(* CODESYS project cr710siowrapper_RECOVERED_2026-03-05T12-49-56.project
   Company: ifm electronic
   Description: Project template with CR711S configured 2.25MByte Standard 2.25MByte Safety
   Title: ifmCR711S_TemplateProject
   Version: 2.4.10.0

Project tree, tasks and I/O mapping:
  StandardPLC : CR710S Standard, ifm electronic, order no. CR710S, version 3.2.0.0
    application Application
      libraries: ifmR360-3, 1.1.1.0 (ifm electronic); Util, * (System); Standard, * (System); CR710S IOWrapper, 1.0.4.9 (ifm electronic)
      task Task (cyclic, interval t#10ms, priority 0) calls PLC_PRG, HeartBeat
      visualisation SimpleStateSwitch
      EVC
      program CR710S_Config [ST]: config_outputs, config_outgroups, config_inputs
      data type EStates
      program PLC_PRG [ST]
      data type EStation
      global variables GVL_HeartBeat
      program HeartBeat [LD]
    HMI : HMI, ifm electronic, version 3.2.0.0
      User_LEDs : User_LEDs, ifm electronic, version 3.2.0.0
          input  UserLED0_I : LED_IEC_B_INPUT_MAPPING_TYPE  // UserLED0_I
          input  UserLED1_I : LED_IEC_B_INPUT_MAPPING_TYPE  // UserLED1_I
          input  UserLED2_I : LED_IEC_B_INPUT_MAPPING_TYPE  // UserLED2_I
          input  UserLED3_I : LED_IEC_B_INPUT_MAPPING_TYPE  // UserLED3_I
          output UserLED0_Q : LED_IEC_B_OUTPUT_MAPPING_TYPE  // User LED 0
          output UserLED1_Q : LED_IEC_B_OUTPUT_MAPPING_TYPE  // User LED 1
          output UserLED2_Q : LED_IEC_B_OUTPUT_MAPPING_TYPE  // User LED 2
          output UserLED3_Q : LED_IEC_B_OUTPUT_MAPPING_TYPE  // User LED 3
    Local_IO : Local_IO, ifm electronic, version 3.2.0.0
      System_Inputs : System_Inputs, ifm electronic, version 3.2.0.0
          input  VBB30 : IN_SYSTEM_VOLTAGE_INPUT_MAPPING_TYPE  // VBB30
          input  VBB15 : IN_SYSTEM_VOLTAGE_INPUT_MAPPING_TYPE  // VBB15
          input  TemperatureBoard0 : IN_TEMPERATURE_INPUT_MAPPING_TYPE  // TemperatureBoard0
          input  TemperatureChip0 : IN_TEMPERATURE_INPUT_MAPPING_TYPE  // TemperatureChip0
      Inputs : Inputs, ifm electronic, version 3.2.0.0
          input  IN0100_I : IN_MULTIFUNCTION_A_INPUT_MAPPING_TYPE  // IN0100_I
          input  IN0101_I : IN_MULTIFUNCTION_A_INPUT_MAPPING_TYPE  // IN0101_I
          input  IN0102_I : IN_MULTIFUNCTION_A_INPUT_MAPPING_TYPE  // IN0102_I
          input  IN0103_I : IN_MULTIFUNCTION_A_INPUT_MAPPING_TYPE  // IN0103_I
          input  IN0600_I : IN_MULTIFUNCTION_A_INPUT_MAPPING_TYPE  // IN0600_I
          input  IN0601_I : IN_MULTIFUNCTION_A_INPUT_MAPPING_TYPE  // IN0601_I
          input  IN0602_I : IN_MULTIFUNCTION_A_INPUT_MAPPING_TYPE  // IN0602_I
          input  IN0603_I : IN_MULTIFUNCTION_A_INPUT_MAPPING_TYPE  // IN0603_I
          input  IN0400_I : IN_RESISTOR_A_INPUT_MAPPING_TYPE  // IN0400_I
          input  IN0401_I : IN_RESISTOR_A_INPUT_MAPPING_TYPE  // IN0401_I
          input  IN0900_I : IN_RESISTOR_A_INPUT_MAPPING_TYPE  // IN0900_I
          input  IN0901_I : IN_RESISTOR_A_INPUT_MAPPING_TYPE  // IN0901_I
          input  COM_RESET_I : IN_COMMUNICATION_RESET_INPUT_MAPPING_TYPE  // COM_RESET_I
          input  IN0000_I : IN_FREQUENCY_B_CHANNEL_A_INPUT_MAPPING_TYPE  // IN0000_I
          input  IN0002_I : IN_FREQUENCY_B_CHANNEL_A_INPUT_MAPPING_TYPE  // IN0002_I
          input  IN0500_I : IN_FREQUENCY_B_CHANNEL_A_INPUT_MAPPING_TYPE  // IN0500_I
          input  IN0502_I : IN_FREQUENCY_B_CHANNEL_A_INPUT_MAPPING_TYPE  // IN0502_I
          input  IN0001_I : IN_FREQUENCY_B_CHANNEL_B_INPUT_MAPPING_TYPE  // IN0001_I
          input  IN0003_I : IN_FREQUENCY_B_CHANNEL_B_INPUT_MAPPING_TYPE  // IN0003_I
          input  IN0501_I : IN_FREQUENCY_B_CHANNEL_B_INPUT_MAPPING_TYPE  // IN0501_I
          input  IN0503_I : IN_FREQUENCY_B_CHANNEL_B_INPUT_MAPPING_TYPE  // IN0503_I
      Outputs : Outputs, ifm electronic, version 3.2.0.0
          input  OUT0006_I : OUT_PWM_40_BRIDGE_A_INPUT_MAPPING_TYPE  // OUT0006_I
          input  OUT0106_I : OUT_PWM_40_BRIDGE_A_INPUT_MAPPING_TYPE  // OUT0106_I
          input  OUT0000_I : OUT_PWM_25_A_INPUT_MAPPING_TYPE  // OUT0000_I
          input  OUT0002_I : OUT_PWM_25_A_INPUT_MAPPING_TYPE  // OUT0002_I
          input  OUT0004_I : OUT_PWM_25_A_INPUT_MAPPING_TYPE  // OUT0004_I
          input  OUT0100_I : OUT_PWM_25_A_INPUT_MAPPING_TYPE  // OUT0100_I
          input  OUT0102_I : OUT_PWM_25_A_INPUT_MAPPING_TYPE  // OUT0102_I
          input  OUT0104_I : OUT_PWM_25_A_INPUT_MAPPING_TYPE  // OUT0104_I
          input  OUT3001_I : OUT_VOLTAGE_A_INPUT_MAPPING_TYPE  // OUT3001_I
          input  OUT3000_I : OUT_SUPPLY_A_INPUT_MAPPING_TYPE  // OUT3000_I
          input  OUT0001_I : OUT_PWM_25_B_INPUT_MAPPING_TYPE  // OUT0001_I
          input  OUT0003_I : OUT_PWM_25_B_INPUT_MAPPING_TYPE  // OUT0003_I
          input  OUT0005_I : OUT_PWM_25_B_INPUT_MAPPING_TYPE  // OUT0005_I
          input  OUT0101_I : OUT_PWM_25_B_INPUT_MAPPING_TYPE  // OUT0101_I
          input  OUT0103_I : OUT_PWM_25_B_INPUT_MAPPING_TYPE  // OUT0103_I
          input  OUT0105_I : OUT_PWM_25_B_INPUT_MAPPING_TYPE  // OUT0105_I
          input  OUT0007_I : OUT_PWM_40_BRIDGE_A_INPUT_MAPPING_TYPE  // OUT0007_I
          input  OUT0107_I : OUT_PWM_40_BRIDGE_A_INPUT_MAPPING_TYPE  // OUT0107_I
          output OUT0006_Q : OUT_PWM_40_BRIDGE_A_OUTPUT_MAPPING_TYPE  // OUT0006_Q
          output OUT0106_Q : OUT_PWM_40_BRIDGE_A_OUTPUT_MAPPING_TYPE  // OUT0106_Q
          output OUT0000_Q : OUT_PWM_25_A_OUTPUT_MAPPING_TYPE  // OUT0000_Q
          output OUT0002_Q : OUT_PWM_25_A_OUTPUT_MAPPING_TYPE  // OUT0002_Q
          output OUT0004_Q : OUT_PWM_25_A_OUTPUT_MAPPING_TYPE  // OUT0004_Q
          output OUT0100_Q : OUT_PWM_25_A_OUTPUT_MAPPING_TYPE  // OUT0100_Q
          output OUT0102_Q : OUT_PWM_25_A_OUTPUT_MAPPING_TYPE  // OUT0102_Q
          output OUT0104_Q : OUT_PWM_25_A_OUTPUT_MAPPING_TYPE  // OUT0104_Q
          output OUT3001_Q : OUT_VOLTAGE_A_OUTPUT_MAPPING_TYPE  // OUT3001_Q
          output OUT3000_Q : OUT_SUPPLY_A_OUTPUT_MAPPING_TYPE  // OUT3000_Q
          output OUT0001_Q : OUT_PWM_25_B_OUTPUT_MAPPING_TYPE  // OUT0001_Q
          output OUT0003_Q : OUT_PWM_25_B_OUTPUT_MAPPING_TYPE  // OUT0003_Q
          output OUT0005_Q : OUT_PWM_25_B_OUTPUT_MAPPING_TYPE  // OUT0005_Q
          output OUT0101_Q : OUT_PWM_25_B_OUTPUT_MAPPING_TYPE  // OUT0101_Q
          output OUT0103_Q : OUT_PWM_25_B_OUTPUT_MAPPING_TYPE  // OUT0103_Q
          output OUT0105_Q : OUT_PWM_25_B_OUTPUT_MAPPING_TYPE  // OUT0105_Q
          output OUT0007_Q : OUT_PWM_40_BRIDGE_A_OUTPUT_MAPPING_TYPE  // OUT0007_Q
          output OUT0107_Q : OUT_PWM_40_BRIDGE_A_OUTPUT_MAPPING_TYPE  // OUT0107_Q
      System_Outputs : System_Outputs, ifm electronic, version 3.2.0.0
          input  VBB0_SW_I : OUT_GROUP_SWITCH_INPUT_MAPPING_TYPE  // VBB0_SW_I
          input  VBB1_SW_I : OUT_GROUP_SWITCH_INPUT_MAPPING_TYPE  // VBB1_SW_I
          output VBB0_SW_Q : OUT_GROUP_SWITCH_OUTPUT_MAPPING_TYPE  // VBB0_SW_Q
          output VBB1_SW_Q : OUT_GROUP_SWITCH_OUTPUT_MAPPING_TYPE  // VBB1_SW_Q
          output SUPPLY_SWITCH_Q : OUT_SYS_SWITCH_OUTPUT_MAPPING_TYPE  // SUPPLY_SWITCH_Q
    Communication : Communication, ifm electronic, version 3.2.0.0
      CAN : CAN, ifm electronic, version 3.2.0.0
      Ethernet : Ethernet, ifm electronic, version 3.2.0.0
  SafetyPLC : CR710S SIL2, ifm electronic, order no. CR710S, version 3.2.0.0
    application Application
      libraries: ifmR360-3, * (ifm electronic); ifmR360-3, 1.1.1.0 (ifm electronic); CR710S IOWrapper, 1.0.4.9 (ifm electronic)
      task Task (cyclic, interval t#10ms, priority 1, watchdog t#8ms x 1) calls PLC_PRG
      program PLC_PRG [ST]
      global variables EVL
    HMI : HMI, ifm electronic, version 3.2.0.0
      User_LEDs : User_LEDs, ifm electronic, version 3.2.0.0
          input  UserLED0_I : LED_IEC_B_INPUT_MAPPING_TYPE  // UserLED0_I
          input  UserLED1_I : LED_IEC_B_INPUT_MAPPING_TYPE  // UserLED1_I
          input  UserLED2_I : LED_IEC_B_INPUT_MAPPING_TYPE  // UserLED2_I
          input  UserLED3_I : LED_IEC_B_INPUT_MAPPING_TYPE  // UserLED3_I
          output UserLED0_Q : LED_IEC_B_OUTPUT_MAPPING_TYPE  // User LED 0
          output UserLED1_Q : LED_IEC_B_OUTPUT_MAPPING_TYPE  // User LED 1
          output UserLED2_Q : LED_IEC_B_OUTPUT_MAPPING_TYPE  // User LED 2
          output UserLED3_Q : LED_IEC_B_OUTPUT_MAPPING_TYPE  // User LED 3
    Local_IO : Local_IO, ifm electronic, version 3.2.0.0
      System_Outputs : System_Outputs, ifm electronic, version 3.2.0.0
          input  VBB0_SW_I : OUT_GROUP_SWITCH_INPUT_MAPPING_TYPE  // VBB0_SW_I
          input  VBB1_SW_I : OUT_GROUP_SWITCH_INPUT_MAPPING_TYPE  // VBB1_SW_I
          output VBB0_SW_Q : OUT_GROUP_SWITCH_OUTPUT_MAPPING_TYPE  // VBB0_SW_Q
          output VBB1_SW_Q : OUT_GROUP_SWITCH_OUTPUT_MAPPING_TYPE  // VBB1_SW_Q
          output SUPPLY_SWITCH_Q : OUT_SYS_SWITCH_OUTPUT_MAPPING_TYPE  // SUPPLY_SWITCH_Q
      Outputs : Outputs, ifm electronic, version 3.2.0.0
          input  OUT0006_I : OUT_PWM_40_BRIDGE_A_INPUT_MAPPING_TYPE  // OUT0006_I
          input  OUT0106_I : OUT_PWM_40_BRIDGE_A_INPUT_MAPPING_TYPE  // OUT0106_I
          input  OUT0000_I : OUT_PWM_25_A_INPUT_MAPPING_TYPE  // OUT0000_I
          input  OUT0002_I : OUT_PWM_25_A_INPUT_MAPPING_TYPE  // OUT0002_I
          input  OUT0004_I : OUT_PWM_25_A_INPUT_MAPPING_TYPE  // OUT0004_I
          input  OUT0100_I : OUT_PWM_25_A_INPUT_MAPPING_TYPE  // OUT0100_I
          input  OUT0102_I : OUT_PWM_25_A_INPUT_MAPPING_TYPE  // OUT0102_I
          input  OUT0104_I : OUT_PWM_25_A_INPUT_MAPPING_TYPE  // OUT0104_I
          input  OUT3001_I : OUT_VOLTAGE_A_INPUT_MAPPING_TYPE  // OUT3001_I
          input  OUT3000_I : OUT_SUPPLY_A_INPUT_MAPPING_TYPE  // OUT3000_I
          input  OUT0001_I : OUT_PWM_25_B_INPUT_MAPPING_TYPE  // OUT0001_I
          input  OUT0003_I : OUT_PWM_25_B_INPUT_MAPPING_TYPE  // OUT0003_I
          input  OUT0005_I : OUT_PWM_25_B_INPUT_MAPPING_TYPE  // OUT0005_I
          input  OUT0101_I : OUT_PWM_25_B_INPUT_MAPPING_TYPE  // OUT0101_I
          input  OUT0103_I : OUT_PWM_25_B_INPUT_MAPPING_TYPE  // OUT0103_I
          input  OUT0105_I : OUT_PWM_25_B_INPUT_MAPPING_TYPE  // OUT0105_I
          input  OUT0007_I : OUT_PWM_40_BRIDGE_A_INPUT_MAPPING_TYPE  // OUT0007_I
          input  OUT0107_I : OUT_PWM_40_BRIDGE_A_INPUT_MAPPING_TYPE  // OUT0107_I
          output OUT0006_Q : OUT_PWM_40_BRIDGE_A_OUTPUT_MAPPING_TYPE  // OUT0006_Q
          output OUT0106_Q : OUT_PWM_40_BRIDGE_A_OUTPUT_MAPPING_TYPE  // OUT0106_Q
          output OUT0000_Q : OUT_PWM_25_A_OUTPUT_MAPPING_TYPE  // OUT0000_Q
          output OUT0002_Q : OUT_PWM_25_A_OUTPUT_MAPPING_TYPE  // OUT0002_Q
          output OUT0004_Q : OUT_PWM_25_A_OUTPUT_MAPPING_TYPE  // OUT0004_Q
          output OUT0100_Q : OUT_PWM_25_A_OUTPUT_MAPPING_TYPE  // OUT0100_Q
          output OUT0102_Q : OUT_PWM_25_A_OUTPUT_MAPPING_TYPE  // OUT0102_Q
          output OUT0104_Q : OUT_PWM_25_A_OUTPUT_MAPPING_TYPE  // OUT0104_Q
          output OUT3001_Q : OUT_VOLTAGE_A_OUTPUT_MAPPING_TYPE  // OUT3001_Q
          output OUT3000_Q : OUT_SUPPLY_A_OUTPUT_MAPPING_TYPE  // OUT3000_Q
          output OUT0001_Q : OUT_PWM_25_B_OUTPUT_MAPPING_TYPE  // OUT0001_Q
          output OUT0003_Q : OUT_PWM_25_B_OUTPUT_MAPPING_TYPE  // OUT0003_Q
          output OUT0005_Q : OUT_PWM_25_B_OUTPUT_MAPPING_TYPE  // OUT0005_Q
          output OUT0101_Q : OUT_PWM_25_B_OUTPUT_MAPPING_TYPE  // OUT0101_Q
          output OUT0103_Q : OUT_PWM_25_B_OUTPUT_MAPPING_TYPE  // OUT0103_Q
          output OUT0105_Q : OUT_PWM_25_B_OUTPUT_MAPPING_TYPE  // OUT0105_Q
          output OUT0007_Q : OUT_PWM_40_BRIDGE_A_OUTPUT_MAPPING_TYPE  // OUT0007_Q
          output OUT0107_Q : OUT_PWM_40_BRIDGE_A_OUTPUT_MAPPING_TYPE  // OUT0107_Q
      System_Inputs : System_Inputs, ifm electronic, version 3.2.0.0
          input  VBB30 : IN_SYSTEM_VOLTAGE_INPUT_MAPPING_TYPE  // VBB30
          input  VBB15 : IN_SYSTEM_VOLTAGE_INPUT_MAPPING_TYPE  // VBB15
          input  TemperatureBoard0 : IN_TEMPERATURE_INPUT_MAPPING_TYPE  // TemperatureBoard0
          input  TemperatureChip0 : IN_TEMPERATURE_INPUT_MAPPING_TYPE  // TemperatureChip0
      Inputs : Inputs, ifm electronic, version 3.2.0.0
          input  IN0100_I : IN_MULTIFUNCTION_A_INPUT_MAPPING_TYPE  // IN0100_I
          input  IN0101_I : IN_MULTIFUNCTION_A_INPUT_MAPPING_TYPE  // IN0101_I
          input  IN0102_I : IN_MULTIFUNCTION_A_INPUT_MAPPING_TYPE  // IN0102_I
          input  IN0103_I : IN_MULTIFUNCTION_A_INPUT_MAPPING_TYPE  // IN0103_I
          input  IN0600_I : IN_MULTIFUNCTION_A_INPUT_MAPPING_TYPE  // IN0600_I
          input  IN0601_I : IN_MULTIFUNCTION_A_INPUT_MAPPING_TYPE  // IN0601_I
          input  IN0602_I : IN_MULTIFUNCTION_A_INPUT_MAPPING_TYPE  // IN0602_I
          input  IN0603_I : IN_MULTIFUNCTION_A_INPUT_MAPPING_TYPE  // IN0603_I
          input  IN0400_I : IN_RESISTOR_A_INPUT_MAPPING_TYPE  // IN0400_I
          input  IN0401_I : IN_RESISTOR_A_INPUT_MAPPING_TYPE  // IN0401_I
          input  IN0900_I : IN_RESISTOR_A_INPUT_MAPPING_TYPE  // IN0900_I
          input  IN0901_I : IN_RESISTOR_A_INPUT_MAPPING_TYPE  // IN0901_I
          input  COM_RESET_I : IN_COMMUNICATION_RESET_INPUT_MAPPING_TYPE  // COM_RESET_I
          input  IN0000_I : IN_FREQUENCY_B_CHANNEL_A_INPUT_MAPPING_TYPE  // IN0000_I
          input  IN0002_I : IN_FREQUENCY_B_CHANNEL_A_INPUT_MAPPING_TYPE  // IN0002_I
          input  IN0500_I : IN_FREQUENCY_B_CHANNEL_A_INPUT_MAPPING_TYPE  // IN0500_I
          input  IN0502_I : IN_FREQUENCY_B_CHANNEL_A_INPUT_MAPPING_TYPE  // IN0502_I
          input  IN0001_I : IN_FREQUENCY_B_CHANNEL_B_INPUT_MAPPING_TYPE  // IN0001_I
          input  IN0003_I : IN_FREQUENCY_B_CHANNEL_B_INPUT_MAPPING_TYPE  // IN0003_I
          input  IN0501_I : IN_FREQUENCY_B_CHANNEL_B_INPUT_MAPPING_TYPE  // IN0501_I
          input  IN0503_I : IN_FREQUENCY_B_CHANNEL_B_INPUT_MAPPING_TYPE  // IN0503_I
    Communication : Communication, ifm electronic, version 3.2.0.0
      Ethernet : Ethernet, ifm electronic, version 3.2.0.0
      CAN : CAN, ifm electronic, version 3.2.0.0
  CR710S : CR710S, ifm electronic, order no. CR710S, version 3.2.0.0
  text list GlobalTextList
*)

// StandardPLC/Application/EStates
{attribute 'qualified_only'}
{attribute 'strict'}
TYPE EStates :
(
	Stable,
	PendingAck, 
	FailSafe 
);
END_TYPE

// StandardPLC/Application/EStation
{attribute 'qualified_only'}
{attribute 'strict'}
TYPE EStation :
(
	Manual, //prio 1
	Remote,  //prio 2
	None
);
END_TYPE

// SafetyPLC/Application/EVL
(* THIS EVL IS AUTOGENERATED. DO NOT MODIFY THESE ATTRIBUTES. *)
{attribute 'location' := '16#800' }
{attribute 'linkalways'}
{attribute 'qualified_only'}
VAR_GLOBAL

END_VAR

// StandardPLC/Application/GVL_HeartBeat
{attribute 'qualified_only'}
VAR_GLOBAL
	HB_Remote_Signal : BOOL;
	HB_Manual_Signal : BOOL;
	
	HB_Remote_OK : BOOL;
	HB_Manual_OK : BOOL;
END_VAR

// SafetyPLC/Application/PLC_PRG
PROGRAM PLC_PRG
VAR
	x : INT;
	y : BOOL; 
END_VAR

END_PROGRAM

// StandardPLC/Application/PLC_PRG
PROGRAM PLC_PRG
VAR

 	// Request takeover
	ReqManual: BOOL; 
	ReqRemote: BOOL; 
	
	// Release control
	RelManual : BOOL;
	RelRemote : BOOL;
	
	//Acknowledge ready
	AckManual: BOOL; 
	AckRemote: BOOL; 
	
	State : EStates; 
	Active : EStation := EStation.Manual; 
	Pending: EStation; 
	
	
	Released : BOOL;
	PendingReady : BOOL;
	
	
	FailSafe: BOOL := FALSE; 
	
	//Granted
	GrantedManual: BOOL; 
	GrantedRemote: BOOL; 
	
	
	Lamp_RequestManual: BOOL; 
	Lamp_RequestRemote: BOOL; 
	Lamp_GrantedManual: BOOL; 
	Lamp_GrantedRemote: BOOL;  
	Lamp_Pending: BOOL;
	
	Lamp_ActiveManual: BOOL;
	Lamp_ActiveRemote: BOOL;
	Lamp_Released: BOOL;
	Lamp_PendingReady: BOOL;
	Lamp_Remote_No_HeartBeat : BOOL;
	Lamp_Manual_No_HeartBeat : BOOL;
	Lamp_FailSafe : BOOL;
	
END_VAR





(*
IOWrapper V1.0.4.4
ifm ecomatic gmbh - VNC - pp 

The licence free software is of average quality and suitable for normal use on common personal
computers. According to the present state of software technology no guarantee can be
assumed for the correct operation or absence of computer viruses nor for the removal of any
fault which may occur. In case of an incorrect program ifm electronic gmbh cannot be held
liable for cost incurred at the customer (e.g. maintenance, repair or rectification of faults).
The exclusion does not apply to damage for which liability is mandatory according to peremptory
legal provisions. Copyright by ifm electronic gmbh, Essen. No copies may be made without the
written permission of ifm electronic gmbh. This also goes for printing images or text for business
use. We reserve the right to make technical alterations.
*)

//CR710S_Config(); 			//IO Configuration

//IOWrapper.READ_INPUTS(); 	//Call IOWrapper Main Program and Read Data from Inputs   

							//Put your Application program here 

//IOWrapper.WRITE_OUTPUTS();	//Call IOWrapper Main Program and Write Data to Outputs 

CASE State OF 
	EStates.Stable: 
		Pending := EStation.None; //No takeover in progress
		IF FailSafe THEN
			Pending := EStation.None;
			State := EStates.Stable;
		
		ELSIF ReqManual AND NOT ReqRemote AND Active <> EStation.Manual AND GVL_HeartBeat.HB_Manual_OK THEN 
			Pending := Estation.Manual;
			State := EStates.PendingAck;

			ELSIF ReqRemote AND NOT ReqManual AND Active <> EStation.Remote AND GVL_HeartBeat.HB_Remote_OK THEN
				Pending := EStation.Remote;
				State := EStates.PendingAck;
		END_IF
	EStates.PendingAck: 
		IF FailSafe THEN
			Pending := EStation.None;
			State := EStates.Stable;
		
		ELSIF (GrantedManual AND (NOT ReqManual OR NOT GVL_HeartBeat.HB_Manual_OK)) OR (GrantedRemote AND (NOT ReqRemote OR NOT GVL_HeartBeat.HB_Remote_OK)) THEN 
			Pending := EStation.None; 
			State := EStates.Stable; 
  
			ELSE
				//Has the current active station released control?
				Released := (Active = EStation.Manual AND RelManual) OR (Active = EStation.Remote AND RelRemote);
		
				// Is the new Pending station ready to take control?
				PendingReady := (Pending = EStation.Manual AND AckManual) OR (Pending = EStation.Remote AND AckRemote);
		
				// Switch only when both are true
				IF Released AND PendingReady THEN
					Active := Pending; 
					Pending := EStation.None;
					State := EStates.Stable;
					//Testar att ta bort dessa
					Released := FALSE; 
					ReqRemote := FALSE; 
					ReqManual := FALSE; 
				END_IF
		END_IF
		
END_CASE

GrantedManual := (Pending = EStation.Manual); 
GrantedRemote := (Pending = EStation.Remote); 


Lamp_RequestManual := ReqManual; 
Lamp_RequestRemote := ReqRemote; 

Lamp_GrantedManual := GrantedManual; 
Lamp_GrantedRemote := GrantedRemote;

Lamp_Pending := (State = EStates.PendingAck); 

Lamp_ActiveManual := (Active = EStation.Manual);
Lamp_ActiveRemote := (Active = EStation.Remote);

Lamp_Released := Released;
Lamp_PendingReady := PendingReady;

Lamp_Remote_No_HeartBeat := ReqRemote AND (NOT GVL_HeartBeat.HB_Remote_OK);
Lamp_Manual_No_HeartBEat := ReqRemote AND (NOT GVL_HeartBeat.HB_Manual_OK);

Lamp_FailSafe := FailSafe;

END_PROGRAM

// StandardPLC/Application/CR710S_Config
PROGRAM CR710S_Config
VAR_INPUT
END_VAR
(*
IOWrapper V1.0.4.3
ifm ecomatic gmbh - VNC - pp 

The licence free software is of average quality and suitable for normal use on common personal
computers. According to the present state of software technology no guarantee can be
assumed for the correct operation or absence of computer viruses nor for the removal of any
fault which may occur. In case of an incorrect program ifm electronic gmbh cannot be held
liable for cost incurred at the customer (e.g. maintenance, repair or rectification of faults).
The exclusion does not apply to damage for which liability is mandatory according to peremptory
legal provisions. Copyright by ifm electronic gmbh, Essen. No copies may be made without the
written permission of ifm electronic gmbh. This also goes for printing images or text for business
use. We reserve the right to make technical alterations.
*)

(* IO Configuration*)
config_inputs();
config_outputs();
config_outgroups();

ACTION config_outputs:
(* Output Mode Configuration *) 
(* Group 0 *)
OUT0000.CONFIG.MONITOR			(FILTER_OUTPUT.UNCHANGED);
OUT0001.CONFIG.MONITOR			(FILTER_OUTPUT.UNCHANGED);
OUT0002.CONFIG.MONITOR			(FILTER_OUTPUT.UNCHANGED);
OUT0003.CONFIG.MONITOR			(FILTER_OUTPUT.UNCHANGED);
OUT0004.CONFIG.MONITOR			(FILTER_OUTPUT.UNCHANGED);
OUT0005.CONFIG.MONITOR			(FILTER_OUTPUT.UNCHANGED);
OUT0006.CONFIG.MONITOR			(FILTER_OUTPUT.UNCHANGED);
OUT0007.CONFIG.MONITOR			(FILTER_OUTPUT.UNCHANGED);
(* Group 1 *)         				    		
OUT0100.CONFIG.MONITOR			(FILTER_OUTPUT.UNCHANGED);
OUT0101.CONFIG.MONITOR			(FILTER_OUTPUT.UNCHANGED);
OUT0102.CONFIG.MONITOR			(FILTER_OUTPUT.UNCHANGED);
OUT0103.CONFIG.MONITOR			(FILTER_OUTPUT.UNCHANGED);
OUT0104.CONFIG.MONITOR			(FILTER_OUTPUT.UNCHANGED);
OUT0105.CONFIG.MONITOR			(FILTER_OUTPUT.UNCHANGED);
OUT0106.CONFIG.MONITOR			(FILTER_OUTPUT.UNCHANGED);
OUT0107.CONFIG.MONITOR			(FILTER_OUTPUT.UNCHANGED);
(* Output SensorSupply and Analogue *)      				
OUT3000.CONFIG.MONITOR			(FILTER_OUTPUT.UNCHANGED);
OUT3001.CONFIG.MONITOR			(FILTER_OUTPUT.UNCHANGED);	

(* Diagnostic and Protection Configuration *) 
(* Group 0 *)
OUT0000.CONFIG.SET_DIAG_LVL_PROT	(0, 2500, 100, eDIAG_PROT_MODE.DIAG_PROT);
OUT0001.CONFIG.SET_DIAG_LVL_PROT	(0, 2500, 100, eDIAG_PROT_MODE.DIAG_PROT);
OUT0002.CONFIG.SET_DIAG_LVL_PROT	(0, 2500, 100, eDIAG_PROT_MODE.DIAG_PROT);
OUT0003.CONFIG.SET_DIAG_LVL_PROT	(0, 2500, 100, eDIAG_PROT_MODE.DIAG_PROT);
OUT0004.CONFIG.SET_DIAG_LVL_PROT	(0, 2500, 100, eDIAG_PROT_MODE.DIAG_PROT);
OUT0005.CONFIG.SET_DIAG_LVL_PROT	(0, 2500, 100, eDIAG_PROT_MODE.DIAG_PROT);
OUT0006.CONFIG.SET_DIAG_LVL_PROT	(0, 4000, 100, eDIAG_PROT_MODE.DIAG_PROT);
OUT0007.CONFIG.SET_DIAG_LVL_PROT	(0, 4000, 100, eDIAG_PROT_MODE.DIAG_PROT);
(* Group 1 *)                                       
OUT0100.CONFIG.SET_DIAG_LVL_PROT	(0, 2500, 100, eDIAG_PROT_MODE.DIAG_PROT);
OUT0101.CONFIG.SET_DIAG_LVL_PROT	(0, 2500, 100, eDIAG_PROT_MODE.DIAG_PROT);
OUT0102.CONFIG.SET_DIAG_LVL_PROT	(0, 2500, 100, eDIAG_PROT_MODE.DIAG_PROT);
OUT0103.CONFIG.SET_DIAG_LVL_PROT	(0, 2500, 100, eDIAG_PROT_MODE.DIAG_PROT);
OUT0104.CONFIG.SET_DIAG_LVL_PROT	(0, 2500, 100, eDIAG_PROT_MODE.DIAG_PROT);
OUT0105.CONFIG.SET_DIAG_LVL_PROT	(0, 2500, 100, eDIAG_PROT_MODE.DIAG_PROT);
OUT0106.CONFIG.SET_DIAG_LVL_PROT	(0, 4000, 100, eDIAG_PROT_MODE.DIAG_PROT);
OUT0107.CONFIG.SET_DIAG_LVL_PROT	(0, 4000, 100, eDIAG_PROT_MODE.DIAG_PROT);
END_ACTION

ACTION config_outgroups:
(* Output Group Mode Configuration *) 
OUTGROUP0.CONFIG.MONITOR				(FILTER_OUTPUT_GROUP.UNCHANGED);
OUTGROUP1.CONFIG.MONITOR				(FILTER_OUTPUT_GROUP.UNCHANGED);

(* Diagnostic and Protection Configuration *) 
OUTGROUP0.CONFIG.SET_DIAG_LVL_PROT		(0, 12000, 100, eDIAG_PROT_MODE.DIAG_PROT);
OUTGROUP1.CONFIG.SET_DIAG_LVL_PROT		(0, 12000, 100, eDIAG_PROT_MODE.DIAG_PROT);
END_ACTION

ACTION config_inputs:
(* Input Mode Configuration *) // FREQ_SENSE_PERIODS.PERIODS_5, ENCODER_RESOLUTION.EVERY_EDGE
(* Frequency Inputs *)
IN0000.CONFIG.MONITOR		(FILTER_INPUT.UNCHANGED);
IN0001.CONFIG.MONITOR		(FILTER_INPUT.UNCHANGED);
IN0002.CONFIG.MONITOR		(FILTER_INPUT.UNCHANGED);
IN0003.CONFIG.MONITOR		(FILTER_INPUT.UNCHANGED);
IN0500.CONFIG.MONITOR		(FILTER_INPUT.UNCHANGED);
IN0501.CONFIG.MONITOR		(FILTER_INPUT.UNCHANGED);
IN0502.CONFIG.MONITOR		(FILTER_INPUT.UNCHANGED);
IN0503.CONFIG.MONITOR		(FILTER_INPUT.UNCHANGED);
(* Multifuntional Inputs *) 
IN0100.CONFIG.MONITOR		(FILTER_INPUT.UNCHANGED);
IN0101.CONFIG.MONITOR		(FILTER_INPUT.UNCHANGED);
IN0102.CONFIG.MONITOR		(FILTER_INPUT.UNCHANGED);
IN0103.CONFIG.MONITOR		(FILTER_INPUT.UNCHANGED);            				
IN0600.CONFIG.MONITOR		(FILTER_INPUT.UNCHANGED);
IN0601.CONFIG.MONITOR		(FILTER_INPUT.UNCHANGED);
IN0602.CONFIG.MONITOR		(FILTER_INPUT.UNCHANGED);
IN0603.CONFIG.MONITOR		(FILTER_INPUT.UNCHANGED);
(* Resistopr Inputs *)      	
IN0400.CONFIG.MONITOR		(FILTER_INPUT.UNCHANGED);
IN0401.CONFIG.MONITOR		(FILTER_INPUT.UNCHANGED);
IN0900.CONFIG.MONITOR		(FILTER_INPUT.UNCHANGED);
IN0901.CONFIG.MONITOR		(FILTER_INPUT.UNCHANGED);

(* Diagnostic and Protection Configuration *) //eDIAG_PROT_MODE.DIAG_PROT
(* Frequency Inputs *) 
IN0000.CONFIG.SET_DIAG_LVL_PROT		(0, 32000, 100, eDIAG_PROT_MODE.DIAG_PROT);
IN0001.CONFIG.SET_DIAG_LVL_PROT		(0, 32000, 100, eDIAG_PROT_MODE.DIAG_PROT);
IN0002.CONFIG.SET_DIAG_LVL_PROT		(0, 32000, 100, eDIAG_PROT_MODE.DIAG_PROT);
IN0003.CONFIG.SET_DIAG_LVL_PROT		(0, 32000, 100, eDIAG_PROT_MODE.DIAG_PROT);
IN0500.CONFIG.SET_DIAG_LVL_PROT		(0, 32000, 100, eDIAG_PROT_MODE.DIAG_PROT);
IN0501.CONFIG.SET_DIAG_LVL_PROT		(0, 32000, 100, eDIAG_PROT_MODE.DIAG_PROT);
IN0502.CONFIG.SET_DIAG_LVL_PROT		(0, 32000, 100, eDIAG_PROT_MODE.DIAG_PROT);
IN0503.CONFIG.SET_DIAG_LVL_PROT		(0, 32000, 100, eDIAG_PROT_MODE.DIAG_PROT);
(* Multifuntional Inputs *)                          
IN0100.CONFIG.SET_DIAG_LVL_PROT		(0, 32000, 100, eDIAG_PROT_MODE.DIAG_PROT);
IN0101.CONFIG.SET_DIAG_LVL_PROT		(0, 32000, 100, eDIAG_PROT_MODE.DIAG_PROT);
IN0102.CONFIG.SET_DIAG_LVL_PROT		(0, 32000, 100, eDIAG_PROT_MODE.DIAG_PROT);
IN0103.CONFIG.SET_DIAG_LVL_PROT		(0, 32000, 100, eDIAG_PROT_MODE.DIAG_PROT);                                                    
IN0600.CONFIG.SET_DIAG_LVL_PROT		(0, 32000, 100, eDIAG_PROT_MODE.DIAG_PROT);
IN0601.CONFIG.SET_DIAG_LVL_PROT		(0, 32000, 100, eDIAG_PROT_MODE.DIAG_PROT);
IN0602.CONFIG.SET_DIAG_LVL_PROT		(0, 32000, 100, eDIAG_PROT_MODE.DIAG_PROT);
IN0603.CONFIG.SET_DIAG_LVL_PROT		(0, 32000, 100, eDIAG_PROT_MODE.DIAG_PROT);
(* Resistopr Inputs *)                               
IN0400.CONFIG.SET_DIAG_LVL_PROT		(0, 32000, 100, eDIAG_PROT_MODE.DIAG_PROT);
IN0401.CONFIG.SET_DIAG_LVL_PROT		(0, 32000, 100, eDIAG_PROT_MODE.DIAG_PROT);
IN0900.CONFIG.SET_DIAG_LVL_PROT		(0, 32000, 100, eDIAG_PROT_MODE.DIAG_PROT);
IN0901.CONFIG.SET_DIAG_LVL_PROT		(0, 32000, 100, eDIAG_PROT_MODE.DIAG_PROT);

(* Digital Switching Threshold - Default ON:= 0.7*Vbb, OFF:= 0.3*Vbb *)
(* Frequency Inputs *) 
IN0000.CONFIG.SET_SWITCH_THRESHOLD(300, 700); // 300 = 30% - 700 = 70%
IN0001.CONFIG.SET_SWITCH_THRESHOLD(300, 700);
IN0002.CONFIG.SET_SWITCH_THRESHOLD(300, 700);
IN0003.CONFIG.SET_SWITCH_THRESHOLD(300, 700);
IN0500.CONFIG.SET_SWITCH_THRESHOLD(300, 700);
IN0501.CONFIG.SET_SWITCH_THRESHOLD(300, 700);
IN0502.CONFIG.SET_SWITCH_THRESHOLD(300, 700);
IN0503.CONFIG.SET_SWITCH_THRESHOLD(300, 700);
(* Multifuntional Inputs *)   
IN0100.CONFIG.SET_SWITCH_THRESHOLD(300, 700);
IN0101.CONFIG.SET_SWITCH_THRESHOLD(300, 700);
IN0102.CONFIG.SET_SWITCH_THRESHOLD(300, 700);
IN0103.CONFIG.SET_SWITCH_THRESHOLD(300, 700);
IN0600.CONFIG.SET_SWITCH_THRESHOLD(300, 700);
IN0601.CONFIG.SET_SWITCH_THRESHOLD(300, 700);
IN0602.CONFIG.SET_SWITCH_THRESHOLD(300, 700);
IN0603.CONFIG.SET_SWITCH_THRESHOLD(300, 700);
(* Resistopr Inputs *)     
IN0400.CONFIG.SET_SWITCH_THRESHOLD(300, 700);
IN0401.CONFIG.SET_SWITCH_THRESHOLD(300, 700);
IN0900.CONFIG.SET_SWITCH_THRESHOLD(300, 700);
IN0901.CONFIG.SET_SWITCH_THRESHOLD(300, 700);
END_ACTION

END_PROGRAM

// StandardPLC/Application/HeartBeat
PROGRAM HeartBeat
VAR
	HB_Remote_Signal : BOOL;
    HB_Manual_Signal : BOOL;

    // Timers
    tHBRemote : TON;
    tHBManual : TON;

    // Output
    HB_Remote_OK : BOOL;
    HB_Manual_OK : BOOL;
END_VAR

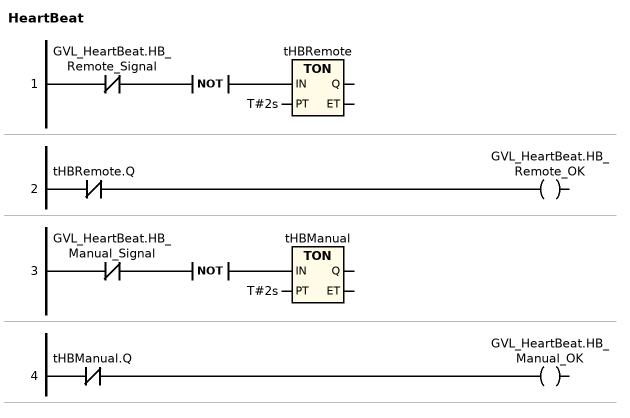
// NETWORK 1
tHBRemote(IN := NOT (NOT GVL_HeartBeat.HB_Remote_Signal), PT := T#2s); // TON

// NETWORK 2
GVL_HeartBeat.HB_Remote_OK := NOT tHBRemote.Q;

// NETWORK 3
tHBManual(IN := NOT (NOT GVL_HeartBeat.HB_Manual_Signal), PT := T#2s); // TON

// NETWORK 4
GVL_HeartBeat.HB_Manual_OK := NOT tHBManual.Q;

END_PROGRAM

// StandardPLC/Application/SimpleStateSwitch
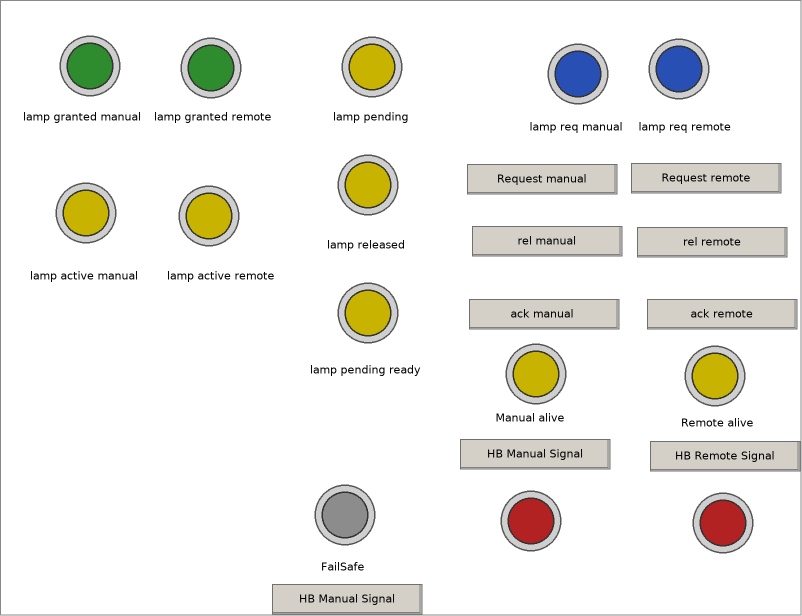
VISUALIZATION SimpleStateSwitch  // 802x616
    Lamp1 (55,31 70x70), variable: PLC_PRG.Lamp_GrantedManual, style: Lamp-Lamp1-Green
    Lamp1 (176,33 70x70), variable: PLC_PRG.Lamp_GrantedRemote, style: Lamp-Lamp1-Green
    Lamp1 (337,32 70x70), variable: PLC_PRG.Lamp_Pending, style: Lamp-Lamp1-Yellow
    Lamp1 (543,39 70x70), variable: PLC_PRG.Lamp_RequestManual, style: Lamp-Lamp1-Blue
    Lamp1 (644,34 70x70), variable: PLC_PRG.Lamp_RequestRemote, style: Lamp-Lamp1-Blue
    Label (9,102 150x30), "lamp granted manual"
    Label (138,102 150x30), "lamp granted remote"
    Label (296,102 150x30), "lamp pending"
    Label (503,112 150x30), "lamp req manual"
    Label (610,112 150x30), "lamp req remote"
    Button (467,164 150x30), "Request manual"
        toggle PLC_PRG.ReqManual
    Button (631,163 150x30), "Request remote"
        toggle PLC_PRG.ReqRemote
    Lamp1 (51,178 70x70), variable: PLC_PRG.Lamp_ActiveManual, style: Lamp-Lamp1-Yellow
    Lamp1 (174,181 70x70), variable: PLC_PRG.Lamp_ActiveRemote, style: Lamp-Lamp1-Yellow
    Label (11,261 150x30), "lamp active manual"
    Label (146,261 150x30), "lamp active remote"
    Lamp1 (333,150 70x70), variable: PLC_PRG.Lamp_Released, style: Lamp-Lamp1-Yellow
    Label (291,230 150x30), "lamp released"
    Lamp1 (333,278 70x70), variable: PLC_PRG.Lamp_PendingReady, style: Lamp-Lamp1-Yellow
    Label (292,355 150x30), "lamp pending ready"
    Button (472,226 150x30), "rel manual"
        toggle PLC_PRG.RelManual
    Button (637,227 150x30), "rel remote"
        toggle PLC_PRG.RelRemote
    Button (469,299 150x30), "ack manual"
        toggle PLC_PRG.AckManual
    Button (647,299 150x30), "ack remote"
        toggle PLC_PRG.AckRemote
    Button (460,439 150x30), "HB Manual Signal"
        toggle GVL_HeartBeat.HB_Manual_Signal
    Button (650,441 150x30), "HB Remote Signal"
        toggle GVL_HeartBeat.HB_Remote_Signal
    Lamp1 (501,339 70x70), variable: GVL_HeartBeat.HB_Manual_OK, style: Lamp-Lamp1-Yellow
    Lamp1 (680,341 70x70), variable: GVL_HeartBeat.HB_Remote_OK, style: Lamp-Lamp1-Yellow
    Label (457,403 150x30), "Manual alive"
    Label (644,408 150x30), "Remote alive"
    Lamp1 (496,486 70x70), variable: PLC_PRG.Lamp_Manual_No_HeartBeat, style: Lamp-Lamp1-Red
    Lamp1 (688,488 70x70), variable: PLC_PRG.Lamp_Remote_No_HeartBeat, style: Lamp-Lamp1-Red
    Lamp1 (310,480 70x70), variable: PLC_PRG.Lamp_FailSafe, style: Lamp-Lamp1-Gray
    Label (268,552 150x30), "FailSafe"
    Button (272,584 150x30), "HB Manual Signal"
        toggle PLC_PRG.FailSafe
END_VISUALIZATION
